# B&R Automation Studio project dbserv_0640 (part 20)

#### dplist.dat
```
;***********************************************************************************
; dplist.dat                                           Erstelldatum:    07.04.2006
; Bearbeiter: 	L.Waibel	                           Letzte Änderung:
;				MEGASYSTEMS Automatisierungssysteme GmbH, München
;***********************************************************************************
"&UST",

"#ALL"
"Client.Anz	=	6",					;Max. Anzahl Clients
"App.Anz	=	6",					;Max. Anzahl Applikationen

;------------------------------------------------------------------------------------------------------------------------
"#BUF"
"Events=10000"						;Anzahl der Ereignisse proDatentypfürLangzeitpufferung
"Typ=0"

;------------------------------------------------------------------------------------------------------------------------
"#TCP",								;Einstellungen für TCP/IP-Treiber
"Client.Timeout = 6000",			;Überwachungszeit
"Client.Port = 20001",				;Ethernet-Port

;------------------------------------------------------------------------------------------------------------------------
"#IEC",								;Einstellungen für IEC-Treiber
"Line=0		IF = IF6.ST1.IF1	MODE =  '/PHY=RS485 /BD=9600 /PA=E /DB=8 /SB=1'"		;Schnittstellenparameter
"Timeout	=	250",				;Überwachungszeit Telegramempfang (in ms)
"Retry.Anz	=	3",					;Wiederholungen bei Telegrammfehlern
"Conn.Anz	=	5",					;Anzahl Anmeldeversuche
"Wait.Intv	= 	60000",				;Wartezeit für Anmeldeversuch (in ms)
"Time.Ts	=   3600000",			;Zeitsyncronisation	(in ms)
"Cmd.Enable	=	1",					;Freigabe Kommandos senden
"Cmd.Timeout=	20000",				;Timeout Empfang von Kommando Rückmeldetelegrammen

;------------------------------------------------------------------------------------------------------------------------
"#L2DP",							;Einstellungen für Profibus-L2DP-Treiber
"Line=0	IF = SS1.IF1 CFG=dpm_099"			; Steckplatz für EX450 / Feldbuskonfiguration
"Timeout	=	1000",				;Überwachungszeit Telegramempfang (in ms)	=1s
"IntvlGrp1	=	1000",				;Zyklus Intervall-Gruppe 1 (in ms)			=1s
"IntvlGrp2	=	60000",				;Zyklus Intervall-Gruppe 2 (in ms)			=1min

;------------------------------------------------------------------------------------------------------------------------
"#VIS"								;Einstellungen für Bedientableau
"Ust.Nr		= 	999",				;Stationsnummer
"Ust.Name	= 	DbsTest",		;Stationsname
;"Ust.IF 	= 	SS1.IF1"			;Schnittstellenparameter für Tableau Büro
"Ust.IF 	= 	SL4.SS1.IF1"		;Schnittstellenparameter für Tableau BMW

;"Grp=1	Name=	SS1_Allgemein"

"TList=1 T0=aus T1=ein"
"TList=2 T0=inaktiv T1=aktiv"
"TList=3 T0=<<< T1=aus T2=ein T3=>>>"
;------------------------------------------------------------------------------------------------------------------------
"#GPS",								;Einstellungen für Funkuhr
									;Achtung! Es kann bis zu 15 Minuten dauern, bis die Satellitenuhr die genaue Position der GPS-Antenne bestimmt hat und sich mit den Atomuhren der Satelliten synchronisiert hat.
"IF.Slot = IF1"				; Schnittstelle für Funkuhr
"IF.Mode = '/PHY=RS485 /PA=N /DB=8 /SB=1 /BD=19200'"	;Modus für Schnittstelle (zur Zeit nur Typ=1 möglich !)
"Tel.Typ = 1"; Meinberg Standard-Zeittelegramm: 				<STX>D:tt.mm.jj;T:w;U:hh.mm.ss;uvxy<ETX>
"Sync.Intv = 1"; Synchronisationsintervall in Minuten
"Tel.Timeout = 30"; Anzahl der Sekunden, nach der einmal eine Warnmeldung erfolgt, wenn kein neues Telegramm eintrifft.
"GPS.Err = GPS_Fehler" 				; Name der Variablen eines anderen Tasks, die im Fehlerfall beschrieben wird
;------------------------------------------------------------------------------------------------------------------------

"$BLOCK",							;Blockdefinitionen für konstante Einträge
"#L2DP Line=0"; ELen=56 ALen=64 Dev.Typ=UMG"
"#I/O Inv=0 Quitt=0"

; ---------------------------
; Datenpunkt-Parametrierungen
; ---------------------------

;"@QUITT"					;Quittierdatenpunkt
;"~Quitt"
;"#ALL Anlage.Nr=1 Typ=QUITT Dp.Nr=1"
;"#I/O ",
;"#VIS ",

;"@KPOS",				;
;"~kpos"
;"#ALL Anlage.Nr=1 Typ=test Dp.Nr=1"
;"#I/O"
;"#VIS Grp=1"

"@IO_7xx0480GSxxx100"
"~W0110 48.0 GSxxx100 "
"#ALL Anlage.Nr=1 Typ=SM Dp.Nr=01"
"#I/O"
"#VIS Grp=1"

; ---------------------------

"@MW_7010480MSA01K01"
"~W0110 48.0 MSA01K01 "
"#ALL Anlage.Nr=1 Typ=MW Dp.Nr=01"
"#I/O"
"#VIS Grp=2"

"@MW_7010480MSA01K02"
"~W0110 48.0 MSA01K02 "
"#ALL Anlage.Nr=2 Typ=MW Dp.Nr=01"
"#I/O"
"#VIS Grp=2"

; ---------------------------

"@MW_7020480MSA02K01"
"~W0110 48.0 MSA02K01 "
"#ALL Anlage.Nr=1 Typ=MW Dp.Nr=02"
"#I/O"
"#VIS Grp=2"

"@MW_7020480MSA02K02"
"~W0110 48.0 MSA02K02 "
"#ALL Anlage.Nr=2 Typ=MW Dp.Nr=02"
"#I/O"
"#VIS Grp=2"

; ---------------------------

"@MW_7030480MSA03K01"
"~W0110 48.0 MSA03K01 "
"#ALL Anlage.Nr=1 Typ=MW Dp.Nr=03"
"#I/O"
"#VIS Grp=2"

"@MW_7030480MSA03K02"
"~W0110 48.0 MSA03K02 "
"#ALL Anlage.Nr=2 Typ=MW Dp.Nr=03"
"#I/O"
"#VIS Grp=2"

; ---------------------------

"@MW_7040480MSA04K01"
"~W0110 48.0 MSA04K01 "
"#ALL Anlage.Nr=1 Typ=MW Dp.Nr=04"
"#I/O"
"#VIS Grp=2"

"@MW_7040480MSA04K02"
"~W0110 48.0 MSA04K02 "
"#ALL Anlage.Nr=2 Typ=MW Dp.Nr=04"
"#I/O"
"#VIS Grp=2"

; ---------------------------

"@MW_7050480MSA05K01"
"~W0110 48.0 MSA05K01 "
"#ALL Anlage.Nr=1 Typ=MW Dp.Nr=05"
"#I/O"
"#VIS Grp=2"

"@MW_7050480MSA05K02"
"~W0110 48.0 MSA05K02 "
"#ALL Anlage.Nr=2 Typ=MW Dp.Nr=05"
"#I/O"
"#VIS Grp=2"

; ---------------------------

"@MW_7060480MSA06K01"
"~W0110 48.0 MSA06K01 "
"#ALL Anlage.Nr=1 Typ=MW Dp.Nr=06"
"#I/O"
"#VIS Grp=2"

"@MW_7060480MSA06K02"
"~W0110 48.0 MSA06K02 "
"#ALL Anlage.Nr=2 Typ=MW Dp.Nr=06"
"#I/O"
"#VIS Grp=2"

; ---------------------------

"@MW_7070480MSA07K01"
"~W0110 48.0 MSA07K01 "
"#ALL Anlage.Nr=1 Typ=MW Dp.Nr=07"
"#I/O"
"#VIS Grp=2"

"@MW_7070480MSA07K02"
"~W0110 48.0 MSA07K02 "
"#ALL Anlage.Nr=2 Typ=MW Dp.Nr=07"
"#I/O"
"#VIS Grp=2"

; ---------------------------

"@MW_7080480MSA08K01"
"~W0110 48.0 MSA08K01 "
"#ALL Anlage.Nr=1 Typ=MW Dp.Nr=08"
"#I/O"
"#VIS Grp=2"

"@MW_7080480MSA08K02"
"~W0110 48.0 MSA08K02 "
"#ALL Anlage.Nr=2 Typ=MW Dp.Nr=08"
"#I/O"
"#VIS Grp=2"

; ---------------------------

"@MW_7100480MSA10K01"
"~W0110 48.0 MSA10K01 "
"#ALL Anlage.Nr=1 Typ=MW Dp.Nr=10"
"#I/O"
"#VIS Grp=2"

"@MW_7100480MSA10K02"
"~W0110 48.0 MSA10K02 "
"#ALL Anlage.Nr=2 Typ=MW Dp.Nr=10"
"#I/O"
"#VIS Grp=2"

; ---------------------------

"@MW_7120480MSA12K01"
"~W0110 48.0 MSA12K01 "
"#ALL Anlage.Nr=1 Typ=MW Dp.Nr=12"
"#I/O"
"#VIS Grp=2"

"@MW_7120480MSA12K02"
"~W0110 48.0 MSA12K02 "
"#ALL Anlage.Nr=2 Typ=MW Dp.Nr=12"
"#I/O"
"#VIS Grp=2"

; ---------------------------

"@MW_7140480MSA14K01"
"~W0110 48.0 MSA14K01 "
"#ALL Anlage.Nr=1 Typ=MW Dp.Nr=14"
"#I/O"
"#VIS Grp=2"

"@MW_7140480MSA14K02"
"~W0110 48.0 MSA14K02 "
"#ALL Anlage.Nr=2 Typ=MW Dp.Nr=14"
"#I/O"
"#VIS Grp=2"

; ---------------------------

"@MW_7160480MSA16K01"
"~W0110 48.0 MSA16K01 "
"#ALL Anlage.Nr=1 Typ=MW Dp.Nr=16"
"#I/O"
"#VIS Grp=2"

"@MW_7160480MSA16K02"
"~W0110 48.0 MSA16K02 "
"#ALL Anlage.Nr=2 Typ=MW Dp.Nr=16"
"#I/O"
"#VIS Grp=2"

; ---------------------------

"@MW_7180480MSA18K01"
"~W0110 48.0 MSA18K01 "
"#ALL Anlage.Nr=1 Typ=MW Dp.Nr=18"
"#I/O"
"#VIS Grp=2"

"@MW_7180480MSA18K02"
"~W0110 48.0 MSA18K02 "
"#ALL Anlage.Nr=2 Typ=MW Dp.Nr=18"
"#I/O"
"#VIS Grp=2"

; ---------------------------

"@MW_7190480MSA19K01"
"~W0110 48.0 MSA19K01 "
"#ALL Anlage.Nr=1 Typ=MW Dp.Nr=19"
"#I/O"
"#VIS Grp=2"

"@MW_7190480MSA19K02"
"~W0110 48.0 MSA19K02 "
"#ALL Anlage.Nr=2 Typ=MW Dp.Nr=19"
"#I/O"
"#VIS Grp=2"

; ---------------------------

"@MW_7500480MSA02K01"
"~W0110 48.0 MSA02K01 "
"#ALL Anlage.Nr=1 Typ=MW Dp.Nr=20"
"#I/O"
"#VIS Grp=2"

; ---------------------------

"@MW_7600480MSA01K01"
"~W0110 48.0 MSA01K01 "
"#ALL Anlage.Nr=1 Typ=MW Dp.Nr=21"
"#I/O"
"#VIS Grp=2"

; ---------------------------

"@MW_7xx0480MSAxxNOT"
"~W0110 48.0 MSAxxNOT "
"#ALL Anlage.Nr=1 Typ=MW Dp.Nr=22"
"#I/O"
"#VIS Grp=2"

; ---------------------------

"@MW_7xx0480MSAxxT01"
"~W0110 48.0 MSAxxT01 "
"#ALL Anlage.Nr=1 Typ=MW Dp.Nr=23"
"#I/O"
"#VIS Grp=2"

; ---------------------------

"@MW_7xx0480MSAxxT02"
"~W0110 48.0 MSAxxT02 "
"#ALL Anlage.Nr=1 Typ=MW Dp.Nr=24"
"#I/O"
"#VIS Grp=2"

; ---------------------------

"@MW_7xx0480MSAxxT03"
"~W0110 48.0 MSAxxT03 "
"#ALL Anlage.Nr=1 Typ=MW Dp.Nr=25"
"#I/O"
"#VIS Grp=2"

; ---------------------------

"@MW_7xx0480MSAxxT04"
"~W0110 48.0 MSAxxT04 "
"#ALL Anlage.Nr=1 Typ=MW Dp.Nr=26"
"#I/O"
"#VIS Grp=2"

; ---------------------------

"@MW_7xx0480MSAxxTEB"
"~W0110 48.0 MSAxxTEB "
"#ALL Anlage.Nr=1 Typ=MW Dp.Nr=27"
"#I/O"
"#VIS Grp=2"

; ---------------------------

"@MW_7xx0480MSAxxK01"
"~W0110 48.0 MSAxxK01 "
"#ALL Anlage.Nr=1 Typ=MW Dp.Nr=28"
"#I/O"
"#VIS Grp=2"

; ---------------------------

"@MW_7xx0480MSAxxK02"
"~W0110 48.0 MSAxxK02 "
"#ALL Anlage.Nr=2 Typ=MW Dp.Nr=20"
"#I/O"
"#VIS Grp=2"

; ---------------------------

"@SPS_7xx0480MSAxxxxxA"
"~W0110 48.0 MSAxxxxx "
"#ALL Anlage.Nr=1 Typ=SPS Dp.Nr=01"
"#I/O"
"#VIS Grp=3"

;--------------------------------------------------------------------------------------
;Feldleitgeräte
"@ABB_015001_MSN01104",				;
"~MSN01104" 									; optionaler Klartext
"#ALL Anlage.Nr=1 Typ=ABB_REF542plus Dp.Nr=1"	; Allgemeine Beschreibung
"#IEC Dev.Adr=104 Line=0 Tsync=1"				; IEC Parametrierung

;--------------------------------------------------------------------------------------
;Sammelschiene 1

"@IO_014001_GSx01100"
"~GSx01100"
"#ALL Anlage.Nr=1 Typ=ALLGMEIN Dp.Nr=01"
"#I/O"
"#VIS Grp=1"

;--------------------------------------------------------------------------------------
;Universalmessgeräte SS1
;"@UMG_013001_USV01100A"
;"~USV01100A"
;"#ALL Anlage.Nr=1 Typ=GSD Dp.Nr=1"
;"#L2DP Dev.Adr=5 Dev.Typ=GSD EAdr=0 Elen=22"
;"#VIS Grp=2"

;"@UMG_013001_USV01100A"
;"~USV01100A"
;"#ALL Anlage.Nr=1 Typ=UMG96 Dp.Nr=1"
;"#L2DP Dev.Adr=1 Dev.Typ=UMGProf EAdr=0 Elen=124 AAdr=0 Alen=2"
;"#VIS Grp=2"

"@UMG_013001_USV01100A"
"~USV01100A"
"#ALL Anlage.Nr=1 Typ=UMG503 Dp.Nr=1"
"#L2DP Line=0 Dev.Adr=1 Dev.Typ=UMG EAdr=0 Elen=56 AAdr=0 Alen=64"
"#VIS Grp=2"
```

### Data object Logical/Anwendung/typlist (Simple, version 0.00.0) - DbServ Datentypliste

- typlist.dat (not shown)

### Program Logical/Anwendung/anlage (IEC) - Musteranlage

#### anlageCyclic.ld - Cyclic code
Diagram, in the editor's own instruction-list form stored in the file:
```il
*******************************************************************
 * COPYRIGHT --
 ********************************************************************
 * Program: anlage
 * File: anlageCyclic.ld
 * Author: waibel
 * Created: August 12, 2013
 ********************************************************************
 * Implementation of program anlage
 *******************************************************************
PROGRAM _CYCLIC

END_PROGRAM
```

#### anlageInit.ld
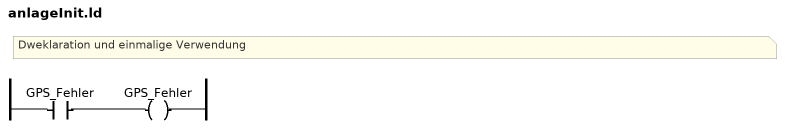
Diagram, in the editor's own instruction-list form stored in the file:
```il
*******************************************************************
 * COPYRIGHT --
 ********************************************************************
 * Program: anlage
 * File: anlageInit.ld
 * Author: waibel
 * Created: August 12, 2013
 ******************************************************************
PROGRAM _INIT

{NetworkNumber := 1}
(* Dweklaration und einmalige Verwendung *)
LD	GPS_Fehler
ST	GPS_Fehler

END_PROGRAM
```

- JAN0926.gsd - GSD-Dateui für UMG503 (not shown)

### Global.var - Globale Variablen
```iecst
(********************************************************************
 * COPYRIGHT --
 ********************************************************************
 * Datei: Global.var
 * Autor: 107044
 * Erstellt: 1. Dezember 2014
 ********************************************************************
 * Globale Variablen des Projekts Impulszaehler
 ********************************************************************)
VAR
	GPS_Fehler : BOOL;
	Impuls_MS1_K1 : UDINT;
	Impuls_MS1_K1_lastMinute : UDINT;
	Impuls_MS1_K1_delta : REAL;
	MW_7010480MSA01K01AMP01 : REAL;
	MW_7010480MSA01K01AZP01 : REAL;
	Impuls_MS1_K2 : UDINT;
	Impuls_MS1_K2_lastMinute : UDINT;
	Impuls_MS1_K2_delta : REAL;
	MW_7010480MSA01K02AMP01 : REAL;
	MW_7010480MSA01K02AZP01 : REAL;
	Impuls_MS2_K1 : UDINT;
	Impuls_MS2_K1_lastMinute : UDINT;
	Impuls_MS2_K1_delta : REAL;
	MW_7020480MSA02K01AMP01 : REAL;
	MW_7020480MSA02K01AZP01 : REAL;
	Impuls_MS2_K2 : UDINT;
	Impuls_MS2_K2_lastMinute : UDINT;
	Impuls_MS2_K2_delta : REAL;
	MW_7020480MSA02K02AMP01 : REAL;
	MW_7020480MSA02K02AZP01 : REAL;
	Impuls_MS3_K1 : UDINT;
	Impuls_MS3_K1_lastMinute : UDINT;
	Impuls_MS3_K1_delta : REAL;
	MW_7030480MSA03K01AMP01 : REAL;
	MW_7030480MSA03K01AZP01 : REAL;
	Impuls_MS3_K2 : UDINT;
	Impuls_MS3_K2_lastMinute : UDINT;
	Impuls_MS3_K2_delta : REAL;
	MW_7030480MSA03K02AMP01 : REAL;
	MW_7030480MSA03K02AZP01 : REAL;
	Impuls_MS4_K1 : UDINT;
	Impuls_MS4_K1_lastMinute : UDINT;
	Impuls_MS4_K1_delta : REAL;
	MW_7040480MSA04K01AMP01 : REAL;
	MW_7040480MSA04K01AZP01 : REAL;
	Impuls_MS4_K2 : UDINT;
	Impuls_MS4_K2_lastMinute : UDINT;
	Impuls_MS4_K2_delta : REAL;
	MW_7040480MSA04K02AMP01 : REAL;
	MW_7040480MSA04K02AZP01 : REAL;
	Impuls_MS5_K1 : UDINT;
	Impuls_MS5_K1_lastMinute : UDINT;
	Impuls_MS5_K1_delta : REAL;
	MW_7050480MSA05K01AMP01 : REAL;
	MW_7050480MSA05K01AZP01 : REAL;
	Impuls_MS5_K2 : UDINT;
	Impuls_MS5_K2_lastMinute : UDINT;
	Impuls_MS5_K2_delta : REAL;
	MW_7050480MSA05K02AMP01 : REAL;
	MW_7050480MSA05K02AZP01 : REAL;
	Impuls_MS6_K1 : UDINT;
	Impuls_MS6_K1_lastMinute : UDINT;
	Impuls_MS6_K1_delta : REAL;
	MW_7060480MSA06K01AMP01 : REAL;
	MW_7060480MSA06K01AZP01 : REAL;
	Impuls_MS6_K2 : UDINT;
	Impuls_MS6_K2_lastMinute : UDINT;
	Impuls_MS6_K2_delta : REAL;
	MW_7060480MSA06K02AMP01 : REAL;
	MW_7060480MSA06K02AZP01 : REAL;
	Impuls_MS7_K1 : UDINT;
	Impuls_MS7_K1_lastMinute : UDINT;
	Impuls_MS7_K1_delta : REAL;
	MW_7070480MSA07K01AMP01 : REAL;
	MW_7070480MSA07K01AZP01 : REAL;
	Impuls_MS7_K2 : UDINT;
	Impuls_MS7_K2_lastMinute : UDINT;
	Impuls_MS7_K2_delta : REAL;
	MW_7070480MSA07K02AMP01 : REAL;
	MW_7070480MSA07K02AZP01 : REAL;
	Impuls_MS8_K1 : UDINT;
	Impuls_MS8_K1_lastMinute : UDINT;
	Impuls_MS8_K1_delta : REAL;
	MW_7080480MSA08K01AMP01 : REAL;
	MW_7080480MSA08K01AZP01 : REAL;
	Impuls_MS8_K2 : UDINT;
	Impuls_MS8_K2_lastMinute : UDINT;
	Impuls_MS8_K2_delta : REAL;
	MW_7080480MSA08K02AMP01 : REAL;
	MW_7080480MSA08K02AZP01 : REAL;
	Impuls_MS10_K1 : UDINT;
	Impuls_MS10_K1_lastMinute : UDINT;
	Impuls_MS10_K1_delta : REAL;
	MW_7100480MSA10K01AMP01 : REAL;
	MW_7100480MSA10K01AZP01 : REAL;
	Impuls_MS10_K2 : UDINT;
	Impuls_MS10_K2_lastMinute : UDINT;
	Impuls_MS10_K2_delta : REAL;
	MW_7100480MSA10K02AMP01 : REAL;
	MW_7100480MSA10K02AZP01 : REAL;
	Impuls_MS12_K1 : UDINT;
	Impuls_MS12_K1_lastMinute : UDINT;
	Impuls_MS12_K1_delta : REAL;
	MW_7120480MSA12K01AMP01 : REAL;
	MW_7120480MSA12K01AZP01 : REAL;
	Impuls_MS12_K2 : UDINT;
	Impuls_MS12_K2_lastMinute : UDINT;
	Impuls_MS12_K2_delta : REAL;
	MW_7120480MSA12K02AMP01 : REAL;
	MW_7120480MSA12K02AZP01 : REAL;
	Impuls_MS14_K1 : UDINT;
	Impuls_MS14_K1_lastMinute : UDINT;
	Impuls_MS14_K1_delta : REAL;
	MW_7140480MSA14K01AMP01 : REAL;
	MW_7140480MSA14K01AZP01 : REAL;
	Impuls_MS14_K2 : UDINT;
	Impuls_MS14_K2_lastMinute : UDINT;
	Impuls_MS14_K2_delta : REAL;
	MW_7140480MSA14K02AMP01 : REAL;
	MW_7140480MSA14K02AZP01 : REAL;
	Impuls_MS16_K1 : UDINT;
	Impuls_MS16_K1_lastMinute : UDINT;
	Impuls_MS16_K1_delta : REAL;
	MW_7160480MSA16K01AMP01 : REAL;
	MW_7160480MSA16K01AZP01 : REAL;
	Impuls_MS16_K2 : UDINT;
	Impuls_MS16_K2_lastMinute : UDINT;
	Impuls_MS16_K2_delta : REAL;
	MW_7160480MSA16K02AMP01 : REAL;
	MW_7160480MSA16K02AZP01 : REAL;
	Impuls_MS18_K1 : UDINT;
	Impuls_MS18_K1_lastMinute : UDINT;
	Impuls_MS18_K1_delta : REAL;
	MW_7180480MSA18K01AMP01 : REAL;
	MW_7180480MSA18K01AZP01 : REAL;
	Impuls_MS18_K2 : UDINT;
	Impuls_MS18_K2_lastMinute : UDINT;
	Impuls_MS18_K2_delta : REAL;
	MW_7180480MSA18K02AMP01 : REAL;
	MW_7180480MSA18K02AZP01 : REAL;
	Impuls_MS19_K1 : UDINT;
	Impuls_MS19_K1_lastMinute : UDINT;
	Impuls_MS19_K1_delta : REAL;
	MW_7190480MSA19K01AMP01 : REAL;
	MW_7190480MSA19K01AZP01 : REAL;
	Impuls_MS19_K2 : UDINT;
	Impuls_MS19_K2_lastMinute : UDINT;
	Impuls_MS19_K2_delta : REAL;
	MW_7190480MSA19K02AMP01 : REAL;
	MW_7190480MSA19K02AZP01 : REAL;
	Impuls_Not_Sued : UDINT;
	Impuls_Not_Sued_lastMinute : UDINT;
	Impuls_Not_Sued_delta : REAL;
	MW_7500480MSA02K01AMP01 : REAL;
	MW_7500480MSA02K01AZP01 : REAL;
	Impuls_Not_Nord : UDINT;
	Impuls_Not_Nord_lastMinute : UDINT;
	Impuls_Not_Nord_delta : REAL;
	MW_7600480MSA01K01AMP01 : REAL;
	MW_7600480MSA01K01AZP01 : REAL;
	Impuls_Not_Station : UDINT;
	Impuls_Not_Station_lastMinute : UDINT;
	Impuls_Not_Station_delta : REAL;
	MW_7xx0480MSAxxNOTAMP01 : REAL;
	MW_7xx0480MSAxxNOTAZP01 : REAL;
	Impuls_Trafo_1 : UDINT;
	Impuls_Trafo_1_lastMinute : UDINT;
	Impuls_Trafo_1_delta : REAL;
	MW_7xx0480MSAxxT01AMP01 : REAL;
	MW_7xx0480MSAxxT01AZP01 : REAL;
	Impuls_Trafo_2 : UDINT;
	Impuls_Trafo_2_lastMinute : UDINT;
	Impuls_Trafo_2_delta : REAL;
	MW_7xx0480MSAxxT02AMP01 : REAL;
	MW_7xx0480MSAxxT02AZP01 : REAL;
	Impuls_Trafo_3 : UDINT;
	Impuls_Trafo_3_lastMinute : UDINT;
	Impuls_Trafo_3_delta : REAL;
	MW_7xx0480MSAxxT03AMP01 : REAL;
	MW_7xx0480MSAxxT03AZP01 : REAL;
	Impuls_Trafo_4 : UDINT;
	Impuls_Trafo_4_lastMinute : UDINT;
	Impuls_Trafo_4_delta : REAL;
	MW_7xx0480MSAxxT04AMP01 : REAL;
	MW_7xx0480MSAxxT04AZP01 : REAL;
	Impuls_EB_Trafo : UDINT;
	Impuls_EB_Trafo_lastMinute : UDINT;
	Impuls_EB_Trafo_delta : REAL;
	MW_7xx0480MSAxxTEBAMP01 : REAL;
	MW_7xx0480MSAxxTEBAZP01 : REAL;
	Impuls_Kabel_1 : UDINT;
	Impuls_Kabel_1_lastMinute : UDINT;
	Impuls_Kabel_1_delta : REAL;
	MW_7xx0480MSAxxK01AMP01 : REAL;
	MW_7xx0480MSAxxK01AZP01 : REAL;
	Impuls_Kabel_2 : UDINT;
	Impuls_Kabel_2_lastMinute : UDINT;
	Impuls_Kabel_2_delta : REAL;
	MW_7xx0480MSAxxK02AMP01 : REAL;
	MW_7xx0480MSAxxK02AZP01 : REAL;
	IO_7xx0480GSxxx100ASM02 : BOOL;
	IO_7xx0480GSxxx100ASM70 : BOOL;
	SPS_7xx0480MSAxxxxxABM98 : BOOL;
	SPS_7xx0480MSAxxxxxABM99 : BOOL;
	TimerWert : BOOL;
	TON_Lebens : TON;
	clock_impuls : TOF;
	clock_pause : TOF;
	clock_rtrig : R_TRIG;
	clock_trigger : BOOL;
END_VAR
```

### Program Logical/zaehler (IEC) - Berechnung Messwerte

#### zaehler.st - Berechnung Messwerte
```iecst
(********************************************************************
 * COPYRIGHT --  Sascha Geißer  --  Kropf Solutions
 ********************************************************************
 * Programm: zaehler
 * Datei: zaehler.st
 * Autor: Sascha Geißer
 * Erstellt: 30. März 2015
 ********************************************************************
 * Berechnung Messwerte
 ********************************************************************)

PROGRAM _INIT

END_PROGRAM

PROGRAM _CYCLIC

	clock_impuls(IN:=NOT clock_pause.Q AND NOT clock_impuls.Q,PT:=t#0s);
	clock_pause(IN:=NOT clock_pause.Q AND NOT clock_impuls.Q,PT:=t#60s);
	clock_rtrig(CLK:=clock_impuls.Q);
	clock_trigger:=clock_rtrig.Q;

	IF clock_trigger THEN

		Impuls_MS1_K1_delta:=UDINT_TO_REAL(Impuls_MS1_K1-Impuls_MS1_K1_lastMinute)*0.4/2;
		MW_7010480MSA01K01AZP01:=MW_7010480MSA01K01AZP01+Impuls_MS1_K1_delta;
		MW_7010480MSA01K01AMP01:=calcMP(Impuls_MS1_K1_delta);
		Impuls_MS1_K1_lastMinute:=Impuls_MS1_K1;

		Impuls_MS1_K2_delta:=UDINT_TO_REAL(Impuls_MS1_K2-Impuls_MS1_K2_lastMinute)*0.4/2;
		MW_7010480MSA01K02AZP01:=MW_7010480MSA01K02AZP01+Impuls_MS1_K2_delta;
		MW_7010480MSA01K02AMP01:=calcMP(Impuls_MS1_K2_delta);
		Impuls_MS1_K2_lastMinute:=Impuls_MS1_K2;

		Impuls_MS2_K1_delta:=UDINT_TO_REAL(Impuls_MS2_K1-Impuls_MS2_K1_lastMinute)*5.0/2;
		MW_7020480MSA02K01AZP01:=MW_7020480MSA02K01AZP01+Impuls_MS2_K1_delta;
		MW_7020480MSA02K01AMP01:=calcMP(Impuls_MS2_K1_delta);
		Impuls_MS2_K1_lastMinute:=Impuls_MS2_K1;

		Impuls_MS2_K2_delta:=UDINT_TO_REAL(Impuls_MS2_K2-Impuls_MS2_K2_lastMinute)*5.0/2;
		MW_7020480MSA02K02AZP01:=MW_7020480MSA02K02AZP01+Impuls_MS2_K2_delta;
		MW_7020480MSA02K02AMP01:=calcMP(Impuls_MS2_K2_delta);
		Impuls_MS2_K2_lastMinute:=Impuls_MS2_K2;

		Impuls_MS3_K1_delta:=UDINT_TO_REAL(Impuls_MS3_K1-Impuls_MS3_K1_lastMinute)*5.0/2;
		MW_7030480MSA03K01AZP01:=MW_7030480MSA03K01AZP01+Impuls_MS3_K1_delta;
		MW_7030480MSA03K01AMP01:=calcMP(Impuls_MS3_K1_delta);
		Impuls_MS3_K1_lastMinute:=Impuls_MS3_K1;

		Impuls_MS3_K2_delta:=UDINT_TO_REAL(Impuls_MS3_K2-Impuls_MS3_K2_lastMinute)*5.0/2;
		MW_7030480MSA03K02AZP01:=MW_7030480MSA03K02AZP01+Impuls_MS3_K2_delta;
		MW_7030480MSA03K02AMP01:=calcMP(Impuls_MS3_K2_delta);
		Impuls_MS3_K2_lastMinute:=Impuls_MS3_K2;

		Impuls_MS4_K1_delta:=UDINT_TO_REAL(Impuls_MS4_K1-Impuls_MS4_K1_lastMinute)*0.6/2;
		MW_7040480MSA04K01AZP01:=MW_7040480MSA04K01AZP01+Impuls_MS4_K1_delta;
		MW_7040480MSA04K01AMP01:=calcMP(Impuls_MS4_K1_delta);
		Impuls_MS4_K1_lastMinute:=Impuls_MS4_K1;

		Impuls_MS4_K2_delta:=UDINT_TO_REAL(Impuls_MS4_K2-Impuls_MS4_K2_lastMinute)*0.6/2;
		MW_7040480MSA04K02AZP01:=MW_7040480MSA04K02AZP01+Impuls_MS4_K2_delta;
		MW_7040480MSA04K02AMP01:=calcMP(Impuls_MS4_K2_delta);
		Impuls_MS4_K2_lastMinute:=Impuls_MS4_K2;

		Impuls_MS5_K1_delta:=UDINT_TO_REAL(Impuls_MS5_K1-Impuls_MS5_K1_lastMinute)*0.6/2;
		MW_7050480MSA05K01AZP01:=MW_7050480MSA05K01AZP01+Impuls_MS5_K1_delta;
		MW_7050480MSA05K01AMP01:=calcMP(Impuls_MS5_K1_delta);
		Impuls_MS5_K1_lastMinute:=Impuls_MS5_K1;

		Impuls_MS5_K2_delta:=UDINT_TO_REAL(Impuls_MS5_K2-Impuls_MS5_K2_lastMinute)*0.6/2;
		MW_7050480MSA05K02AZP01:=MW_7050480MSA05K02AZP01+Impuls_MS5_K2_delta;
		MW_7050480MSA05K02AMP01:=calcMP(Impuls_MS5_K2_delta);
		Impuls_MS5_K2_lastMinute:=Impuls_MS5_K2;

		Impuls_MS6_K1_delta:=UDINT_TO_REAL(Impuls_MS6_K1-Impuls_MS6_K1_lastMinute)*0.4/2;
		MW_7060480MSA06K01AZP01:=MW_7060480MSA06K01AZP01+Impuls_MS6_K1_delta;
		MW_7060480MSA06K01AMP01:=calcMP(Impuls_MS6_K1_delta);
		Impuls_MS6_K1_lastMinute:=Impuls_MS6_K1;

		Impuls_MS6_K2_delta:=UDINT_TO_REAL(Impuls_MS6_K2-Impuls_MS6_K2_lastMinute)*0.4/2;
		MW_7060480MSA06K02AZP01:=MW_7060480MSA06K02AZP01+Impuls_MS6_K2_delta;
		MW_7060480MSA06K02AMP01:=calcMP(Impuls_MS6_K2_delta);
		Impuls_MS6_K2_lastMinute:=Impuls_MS6_K2;

		Impuls_MS7_K1_delta:=UDINT_TO_REAL(Impuls_MS7_K1-Impuls_MS7_K1_lastMinute)*0.4/2;
		MW_7070480MSA07K01AZP01:=MW_7070480MSA07K01AZP01+Impuls_MS7_K1_delta;
		MW_7070480MSA07K01AMP01:=calcMP(Impuls_MS7_K1_delta);
		Impuls_MS7_K1_lastMinute:=Impuls_MS7_K1;

		Impuls_MS7_K2_delta:=UDINT_TO_REAL(Impuls_MS7_K2-Impuls_MS7_K2_lastMinute)*0.4/2;
		MW_7070480MSA07K02AZP01:=MW_7070480MSA07K02AZP01+Impuls_MS7_K2_delta;
		MW_7070480MSA07K02AMP01:=calcMP(Impuls_MS7_K2_delta);
		Impuls_MS7_K2_lastMinute:=Impuls_MS7_K2;

		Impuls_MS8_K1_delta:=UDINT_TO_REAL(Impuls_MS8_K1-Impuls_MS8_K1_lastMinute)*0.6/2;
		MW_7080480MSA08K01AZP01:=MW_7080480MSA08K01AZP01+Impuls_MS8_K1_delta;
		MW_7080480MSA08K01AMP01:=calcMP(Impuls_MS8_K1_delta);
		Impuls_MS8_K1_lastMinute:=Impuls_MS8_K1;

		Impuls_MS8_K2_delta:=UDINT_TO_REAL(Impuls_MS8_K2-Impuls_MS8_K2_lastMinute)*0.6/2;
		MW_7080480MSA08K02AZP01:=MW_7080480MSA08K02AZP01+Impuls_MS8_K2_delta;
		MW_7080480MSA08K02AMP01:=calcMP(Impuls_MS8_K2_delta);
		Impuls_MS8_K2_lastMinute:=Impuls_MS8_K2;

		Impuls_MS10_K1_delta:=UDINT_TO_REAL(Impuls_MS10_K1-Impuls_MS10_K1_lastMinute)*0.6/2;
		MW_7100480MSA10K01AZP01:=MW_7100480MSA10K01AZP01+Impuls_MS10_K1_delta;
		MW_7100480MSA10K01AMP01:=calcMP(Impuls_MS10_K1_delta);
		Impuls_MS10_K1_lastMinute:=Impuls_MS10_K1;

		Impuls_MS10_K2_delta:=UDINT_TO_REAL(Impuls_MS10_K2-Impuls_MS10_K2_lastMinute)*0.6/2;
		MW_7100480MSA10K02AZP01:=MW_7100480MSA10K02AZP01+Impuls_MS10_K2_delta;
		MW_7100480MSA10K02AMP01:=calcMP(Impuls_MS10_K2_delta);
		Impuls_MS10_K2_lastMinute:=Impuls_MS10_K2;

		Impuls_MS12_K1_delta:=UDINT_TO_REAL(Impuls_MS12_K1-Impuls_MS12_K1_lastMinute)*0.4/2;
		MW_7120480MSA12K01AZP01:=MW_7120480MSA12K01AZP01+Impuls_MS12_K1_delta;
		MW_7120480MSA12K01AMP01:=calcMP(Impuls_MS12_K1_delta);
		Impuls_MS12_K1_lastMinute:=Impuls_MS12_K1;

		Impuls_MS12_K2_delta:=UDINT_TO_REAL(Impuls_MS12_K2-Impuls_MS12_K2_lastMinute)*0.4/2;
		MW_7120480MSA12K02AZP01:=MW_7120480MSA12K02AZP01+Impuls_MS12_K2_delta;
		MW_7120480MSA12K02AMP01:=calcMP(Impuls_MS12_K2_delta);
		Impuls_MS12_K2_lastMinute:=Impuls_MS12_K2;

		Impuls_MS14_K1_delta:=UDINT_TO_REAL(Impuls_MS14_K1-Impuls_MS14_K1_lastMinute)*0.6/2;
		MW_7140480MSA14K01AZP01:=MW_7140480MSA14K01AZP01+Impuls_MS14_K1_delta;
		MW_7140480MSA14K01AMP01:=calcMP(Impuls_MS14_K1_delta);
		Impuls_MS14_K1_lastMinute:=Impuls_MS14_K1;

		Impuls_MS14_K2_delta:=UDINT_TO_REAL(Impuls_MS14_K2-Impuls_MS14_K2_lastMinute)*0.6/2;
		MW_7140480MSA14K02AZP01:=MW_7140480MSA14K02AZP01+Impuls_MS14_K2_delta;
		MW_7140480MSA14K02AMP01:=calcMP(Impuls_MS14_K2_delta);
		Impuls_MS14_K2_lastMinute:=Impuls_MS14_K2;

		Impuls_MS16_K1_delta:=UDINT_TO_REAL(Impuls_MS16_K1-Impuls_MS16_K1_lastMinute)*0.4/2;
		MW_7160480MSA16K01AZP01:=MW_7160480MSA16K01AZP01+Impuls_MS16_K1_delta;
		MW_7160480MSA16K01AMP01:=calcMP(Impuls_MS16_K1_delta);
		Impuls_MS16_K1_lastMinute:=Impuls_MS16_K1;

		Impuls_MS16_K2_delta:=UDINT_TO_REAL(Impuls_MS16_K2-Impuls_MS16_K2_lastMinute)*0.4/2;
		MW_7160480MSA16K02AZP01:=MW_7160480MSA16K02AZP01+Impuls_MS16_K2_delta;
		MW_7160480MSA16K02AMP01:=calcMP(Impuls_MS16_K2_delta);
		Impuls_MS16_K2_lastMinute:=Impuls_MS16_K2;

		Impuls_MS18_K1_delta:=UDINT_TO_REAL(Impuls_MS18_K1-Impuls_MS18_K1_lastMinute)*0.4/2;
		MW_7180480MSA18K01AZP01:=MW_7180480MSA18K01AZP01+Impuls_MS18_K1_delta;
		MW_7180480MSA18K01AMP01:=calcMP(Impuls_MS18_K1_delta);
		Impuls_MS18_K1_lastMinute:=Impuls_MS18_K1;

		Impuls_MS18_K2_delta:=UDINT_TO_REAL(Impuls_MS18_K2-Impuls_MS18_K2_lastMinute)*0.4/2;
		MW_7180480MSA18K02AZP01:=MW_7180480MSA18K02AZP01+Impuls_MS18_K2_delta;
		MW_7180480MSA18K02AMP01:=calcMP(Impuls_MS18_K2_delta);
		Impuls_MS18_K2_lastMinute:=Impuls_MS18_K2;

		Impuls_MS19_K1_delta:=UDINT_TO_REAL(Impuls_MS19_K1-Impuls_MS19_K1_lastMinute)*0.3/2;
		MW_7190480MSA19K01AZP01:=MW_7190480MSA19K01AZP01+Impuls_MS19_K1_delta;
		MW_7190480MSA19K01AMP01:=calcMP(Impuls_MS19_K1_delta);
		Impuls_MS19_K1_lastMinute:=Impuls_MS19_K1;

		Impuls_MS19_K2_delta:=UDINT_TO_REAL(Impuls_MS19_K2-Impuls_MS19_K2_lastMinute)*0.3/2;
		MW_7190480MSA19K02AZP01:=MW_7190480MSA19K02AZP01+Impuls_MS19_K2_delta;
		MW_7190480MSA19K02AMP01:=calcMP(Impuls_MS19_K2_delta);
		Impuls_MS19_K2_lastMinute:=Impuls_MS19_K2;

		Impuls_Not_Sued_delta:=UDINT_TO_REAL(Impuls_Not_Sued-Impuls_Not_Sued_lastMinute)*0.3/2;
		MW_7500480MSA02K01AZP01:=MW_7500480MSA02K01AZP01+Impuls_Not_Sued_delta;
		MW_7500480MSA02K01AMP01:=calcMP(Impuls_Not_Sued_delta);
		Impuls_Not_Sued_lastMinute:=Impuls_Not_Sued;

		Impuls_Not_Nord_delta:=UDINT_TO_REAL(Impuls_Not_Nord-Impuls_Not_Nord_lastMinute)*0.3/2;
		MW_7600480MSA01K01AZP01:=MW_7600480MSA01K01AZP01+Impuls_Not_Nord_delta;
		MW_7600480MSA01K01AMP01:=calcMP(Impuls_Not_Nord_delta);
		Impuls_Not_Nord_lastMinute:=Impuls_Not_Nord;

		Impuls_Not_Station_delta:=UDINT_TO_REAL(Impuls_Not_Station-Impuls_Not_Station_lastMinute)*0.3/2;
		MW_7xx0480MSAxxNOTAZP01:=MW_7xx0480MSAxxNOTAZP01+Impuls_Not_Station_delta;
		MW_7xx0480MSAxxNOTAMP01:=calcMP(Impuls_Not_Station_delta);
		Impuls_Not_Station_lastMinute:=Impuls_Not_Station;

		Impuls_Trafo_1_delta:=UDINT_TO_REAL(Impuls_Trafo_1-Impuls_Trafo_1_lastMinute)*3.3/2;
		MW_7xx0480MSAxxT01AZP01:=MW_7xx0480MSAxxT01AZP01+Impuls_Trafo_1_delta;
		MW_7xx0480MSAxxT01AMP01:=calcMP(Impuls_Trafo_1_delta);
		Impuls_Trafo_1_lastMinute:=Impuls_Trafo_1;

		Impuls_Trafo_2_delta:=UDINT_TO_REAL(Impuls_Trafo_2-Impuls_Trafo_2_lastMinute)*3.3/2;
		MW_7xx0480MSAxxT02AZP01:=MW_7xx0480MSAxxT02AZP01+Impuls_Trafo_2_delta;
		MW_7xx0480MSAxxT02AMP01:=calcMP(Impuls_Trafo_2_delta);
		Impuls_Trafo_2_lastMinute:=Impuls_Trafo_2;

		Impuls_Trafo_3_delta:=UDINT_TO_REAL(Impuls_Trafo_3-Impuls_Trafo_3_lastMinute)*3.3/2;
		MW_7xx0480MSAxxT03AZP01:=MW_7xx0480MSAxxT03AZP01+Impuls_Trafo_3_delta;
		MW_7xx0480MSAxxT03AMP01:=calcMP(Impuls_Trafo_3_delta);
		Impuls_Trafo_3_lastMinute:=Impuls_Trafo_3;

		Impuls_Trafo_4_delta:=UDINT_TO_REAL(Impuls_Trafo_4-Impuls_Trafo_4_lastMinute)*3.3/2;
		MW_7xx0480MSAxxT04AZP01:=MW_7xx0480MSAxxT04AZP01+Impuls_Trafo_4_delta;
		MW_7xx0480MSAxxT04AMP01:=calcMP(Impuls_Trafo_4_delta);
		Impuls_Trafo_4_lastMinute:=Impuls_Trafo_4;

		Impuls_EB_Trafo_delta:=UDINT_TO_REAL(Impuls_EB_Trafo-Impuls_EB_Trafo_lastMinute)*0.1/2;
		MW_7xx0480MSAxxTEBAZP01:=MW_7xx0480MSAxxTEBAZP01+Impuls_EB_Trafo_delta;
		MW_7xx0480MSAxxTEBAMP01:=calcMP(Impuls_EB_Trafo_delta);
		Impuls_EB_Trafo_lastMinute:=Impuls_EB_Trafo;

		Impuls_Kabel_1_delta:=UDINT_TO_REAL(Impuls_Kabel_1-Impuls_Kabel_1_lastMinute)*10/2;
		MW_7xx0480MSAxxK01AZP01:=MW_7xx0480MSAxxK01AZP01+Impuls_Kabel_1_delta;
		MW_7xx0480MSAxxK01AMP01:=calcMP(Impuls_Kabel_1_delta);
		Impuls_Kabel_1_lastMinute:=Impuls_Kabel_1;

		Impuls_Kabel_2_delta:=UDINT_TO_REAL(Impuls_Kabel_2-Impuls_Kabel_2_lastMinute)*10/2;
		MW_7xx0480MSAxxK02AZP01:=MW_7xx0480MSAxxK02AZP01+Impuls_Kabel_2_delta;
		MW_7xx0480MSAxxK02AMP01:=calcMP(Impuls_Kabel_2_delta);
		Impuls_Kabel_2_lastMinute:=Impuls_Kabel_2;

	END_IF;

END_PROGRAM
```

#### calcMP.st - Berechnung Wirkleistung
```iecst
(********************************************************************
 * COPYRIGHT --  Sascha Geißer  --  Kropf Solutions
 ********************************************************************
 * Programm: zaehler
 * Datei: calcMP.st
 * Autor: Sascha Geißer
 * Erstellt: 30. März 2015
 ********************************************************************
 * Berechnung Wirkleistung
 ********************************************************************)

FUNCTION calcMP
	calcMP:=Wirkarbeit*60;
END_FUNCTION
```

#### zaehler.fun
```iecst
(********************************************************************
 * COPYRIGHT --  Sascha Geißer  --  Kropf Solutions
 ********************************************************************
 * Programm: zaehler
 * Datei: zaehler.fun
 * Autor: Sascha Geißer
 * Erstellt: 30. März 2015
 ********************************************************************
 * Funktionen und Funktionsblöcke des Programmes zaehler
 ********************************************************************)

FUNCTION calcMP : REAL (*Berechnung Wirkleistung*)
	VAR_INPUT
		Wirkarbeit : REAL;
	END_VAR
END_FUNCTION
```

### Program Logical/Lebensbit (IEC) - Ein neues Programm

#### Lebensbit.st - Zyklischer Code
```iecst
PROGRAM _CYCLIC

	TON_Lebens(IN :=SPS_7xx0480MSAxxxxxABM99 , PT :=t#10s );
	TimerWert:=TON_Lebens.Q;

	IF(TimerWert=TRUE)
		THEN
			SPS_7xx0480MSAxxxxxABM99:=FALSE;
	END_IF

	SPS_7xx0480MSAxxxxxABM98:=SPS_7xx0480MSAxxxxxABM99;

END_PROGRAM
```

### Program Logical/ident (IEC) - Identifikation

#### ident.ab - Zyklischer Code
```automation-basic
(* Identifikation SPS-Programm *)

; SuMSE W0110_Impuls_G0480_O3
; Türnummer:

; NSI:
; IP-Adresse:
; Subnet:
; Gateway:

; Automation Studio Version 3.0.90.31
```

### Program Logical/def (IEC) - Variablendefinition

#### def.st - Zyklischer Code
```iecst
(********************************************************************
 * COPYRIGHT --
 ********************************************************************
 * Programm: def
 * Datei: def.st
 * Autor: 107044
 * Erstellt: 31. März 2015
 ********************************************************************
 * Implementierung des Programms def
 ********************************************************************)

PROGRAM _CYCLIC

	IO_7xx0480GSxxx100ASM02;
	IO_7xx0480GSxxx100ASM70;

END_PROGRAM
```

Listed in the project but not available here: Logical/GlobalIncludes/dbsfunc.c, Logical/GlobalIncludes/bksysall.c, Logical/GlobalIncludes/parser.c, Logical/DbServ-Basis/dbsmon/dbsfunc.c, Logical/DbServ-Basis/dbsevent/dbsfunc.c, Logical/DbServ-Basis/dbslib/bksysall.c, Logical/DbServ-Basis/dbstcp/dbsfunc.c, Logical/GlobalIncludes/parser.c, Logical/GlobalIncludes/bksysall.c, Logical/GlobalIncludes/dbsfunc.c, Logical/IEC103-Treiber/iec103Cmd/Types.typ, Logical/GlobalIncludes/parser.c, Logical/GlobalIncludes/dbsfunc.c, Logical/GlobalIncludes/bksysall.c
